FUNCTION_BLOCK FB_SingleTankS
VAR
	sName : STRING;
	sWeightUnit : STRING := 'Kg'; // Kg
	poCylinderCoil : FB_DigitalOutput;
END_VAR

PROPERTY Name : String
GET
Name := sName;
END_GET
SET
sName := Name;
END_SET
END_PROPERTY

PROPERTY Ref_poCylinderCoil : REFERENCE TO FB_DigitalOutput
GET
Ref_poCylinderCoil ref= poCylinderCoil;
END_GET
END_PROPERTY

PROPERTY WeightUnit : string
GET
WeightUnit := sWeightUnit;
END_GET
SET
sWeightUnit := WeightUnit;
END_SET
END_PROPERTY

END_FUNCTION_BLOCK

(* stored: Version 1.1.0.1, ProductVersion 3.1.4024.12
   POU FB_SingleTankS: Id {c7011563-99b7-45b6-b83f-55dad7d158a9}, SpecialFunc None
   Property Name: Id {05a44893-0e59-489c-ab37-c2b76ac25e38}
   Get Get: Id {9eea58d6-0334-4998-9031-5aa22dfc47f6}
   Set Set: Id {7433cae2-48e3-4de8-9882-cf404880d6c2}
   Property Ref_poCylinderCoil: Id {3e6c3b91-e427-46ec-8253-fffb1f49c5c1}
   Get Get: Id {95935c6d-9b52-48c7-84ee-804067a2c5a8}
   Property WeightUnit: Id {8f2e128a-8c3a-4e4f-81e2-94b76d011fc3}
   Get Get: Id {582dd959-d475-4cc5-b556-b55efd9c8171}
   Set Set: Id {3859c695-f8c1-4be5-b4e1-50beb66e9aa2} *)
